// TwinCAT 3 PLC project LightSwitch
// ProgramVersion: 3.1.4023.0
// libraries:
//   Tc2_Standard, * (Beckhoff Automation GmbH)
//   Tc2_System, * (Beckhoff Automation GmbH)
//   Tc3_Module, * (Beckhoff Automation GmbH)
// project tree:
//   / PlcTask.TcTTO
//   POUs/Customer/ FB_LightController.TcPOU
//   POUs/Lib/ FB_LightBase.TcPOU, FB_LightDimmable.TcPOU, FB_LightGroup.TcPOU, I_LightBase.TcIO, I_LightDimmable.TcIO
//   POUs/ MAIN.TcPOU
// real-time tasks:
//   TASK PlcTask1: cycle T#10ms, priority 21, ADS port 351

CONFIGURATION LightSwitch
    RESOURCE PLC ON TwinCAT3
        TASK PlcTask(INTERVAL := T#10ms, PRIORITY := 21);
        PROGRAM MAIN WITH PlcTask : MAIN;
    END_RESOURCE
END_CONFIGURATION

// ---- POUs/Lib/I_LightBase.TcIO
INTERFACE I_LightBase EXTENDS __SYSTEM.IQueryInterface

PROPERTY ID : USINT
GET
END_GET
SET
END_SET
END_PROPERTY

PROPERTY PUBLIC State : BOOL
GET
END_GET
SET
END_SET
END_PROPERTY

METHOD Toggle
END_METHOD

METHOD TurnOFF
END_METHOD

METHOD TurnON
END_METHOD

END_INTERFACE

// ---- POUs/Lib/I_LightDimmable.TcIO
INTERFACE I_LightDimmable EXTENDS I_LightBase

PROPERTY Brightness : USINT
GET
END_GET
SET
END_SET
END_PROPERTY

END_INTERFACE

// ---- POUs/MAIN.TcPOU
PROGRAM MAIN
VAR
	fbLightController	: FB_LightController;
END_VAR
VAR CONSTANT
	MAXIMUM_NUMBER_OF_LIGHTS	: USINT := 8;
END_VAR

fbLightController();

END_PROGRAM

// ---- POUs/Customer/FB_LightController.TcPOU
FUNCTION_BLOCK FB_LightController
VAR
	_iLight									: I_LightBase;
	_iLightB								: I_LightDimmable;
	                    	    			
	fbLightGroup							: FB_LightGroup;
	                    	    			
	fbLightBase_1							: FB_LightBase;
	fbLightBase_2							: FB_LightBase;
	fbLightBase_3							: FB_LightBase;
	fbLightBase_4							: FB_LightBase;
	fbLightDimmable_5						: FB_LightDimmable;
	fbLightDimmable_6						: FB_LightDimmable;
	fbLightDimmable_7						: FB_LightDimmable;
	fbLightDimmable_8						: FB_LightDimmable;
	                    	    			
	nBrightness								: USINT := 100;
	                    	    			
	bToggle									: BOOL;
	bSwitch									: BOOL;
	bSetBrightness							: BOOL;
	                    	    			
	tToggle									: R_TRIG;
	tSwitchON								: R_TRIG;
	tSwitchOFF								: F_TRIG;
	tSetBrightness							: R_TRIG;
	                    	    			
	bGroupSwitch							: BOOL;
	bSetGroupBrightness						: BOOL;
	                    	    			
	tGroupSwitchON							: R_TRIG;
	tGroupSwitchOFF							: F_TRIG;
	tSetGroupBrightness						: R_TRIG;
	                    	    			
	eSwitchOptions							: (WAIT, TOGGLE, SWITCHON, SWITCHOFF, SETBRIGHTNESS, GROUPSWITCHON, GROUPSWITCHOFF, SETGROUPBRIGHTNESS);
	
	eSwitchControlledLightObjectByLightID	: (LIGHT_ONE, LIGHT_TWO, LIGHT_THREE, LIGHT_FOUR, LIGHT_FIVE, LIGHT_SIX, LIGHT_SEVEN, LIGHT_EIGHT);

END_VAR

fbLightGroup();

CASE eSwitchOptions OF
	WAIT:
		//do nothing
	TOGGLE:
		_iLight.Toggle();
		eSwitchOptions := WAIT;
	SWITCHON:
		_iLight.TurnON();
		eSwitchOptions := WAIT;
	SWITCHOFF:
		_iLight.TurnOFF();
		eSwitchOptions := WAIT;
	SETBRIGHTNESS:
		IF __QUERYINTERFACE(_iLight, _iLightB) THEN
			_iLightB.Brightness := nBrightness;	
		END_IF
		eSwitchOptions := WAIT;
	GROUPSWITCHON:
		fbLightGroup.TurnON();
		eSwitchOptions := WAIT;
	GROUPSWITCHOFF:
		fbLightGroup.TurnOFF();
		eSwitchOptions := WAIT;
	SETGROUPBRIGHTNESS:
		fbLightGroup.SetBrightness(nBrightness);
		eSwitchOptions := WAIT;
END_CASE

CASE eSwitchControlledLightObjectByLightID OF
	LIGHT_ONE:
		ipLight := fbLightBase_1;
	LIGHT_TWO:
		ipLight := fbLightBase_2;
	LIGHT_THREE:
		ipLight := fbLightBase_3;
	LIGHT_FOUR:
		ipLight := fbLightBase_4;
	LIGHT_FIVE:
		ipLight := fbLightDimmable_5;
	LIGHT_SIX:
		ipLight := fbLightDimmable_6;
	LIGHT_SEVEN:
		ipLight := fbLightDimmable_7;
	LIGHT_EIGHT:
		ipLight := fbLightDimmable_8;
END_CASE

tToggle(CLK := bToggle);
tSwitchON(CLK := bSwitch);
tSwitchOFF(CLK := bSwitch);
tSetBrightness(CLK := bSetBrightness);

tGroupSwitchOFF(CLK := bGroupSwitch);
tGroupSwitchON(CLK := bGroupSwitch);
tSetGroupBrightness(CLK := bSetGroupBrightness);

IF tToggle.Q THEN
	eSwitchOptions := TOGGLE;
	bToggle := FALSE;									
END_IF

IF tSwitchON.Q THEN
	eSwitchOptions := SWITCHON;
END_IF

IF tSwitchOFF.Q THEN
	eSwitchOptions := SWITCHOFF;
END_IF

IF tSetBrightness.Q THEN
	eSwitchOptions := SETBRIGHTNESS;
	bSetBrightness := FALSE;
END_IF

IF tGroupSwitchON.Q THEN
	eSwitchOptions := GROUPSWITCHON;
END_IF

IF tGroupSwitchOFF.Q THEN
	eSwitchOptions := GROUPSWITCHOFF;
END_IF

IF tSetGroupBrightness.Q THEN
	eSwitchOptions := SETGROUPBRIGHTNESS;
	bSetGroupBrightness := FALSE;
END_IF

METHOD FB_init : BOOL
VAR_INPUT
	bInitRetains	: BOOL; // if TRUE, the retain variables are initialized (warm start / cold start)
	bInCopyCode		: BOOL;  // if TRUE, the instance afterwards gets moved into the copy code (online change)
END_VAR
_iLight := fbLightBase_1;

fbLightGroup.ImportLight(fbLightBase_1);
fbLightGroup.ImportLight(fbLightBase_2);
fbLightGroup.ImportLight(fbLightBase_3);
fbLightGroup.ImportLight(fbLightBase_4);
fbLightGroup.ImportLight(fbLightDimmable_5);
fbLightGroup.ImportLight(fbLightDimmable_6);
fbLightGroup.ImportLight(fbLightDimmable_7);
fbLightGroup.ImportLight(fbLightDimmable_8);
END_METHOD

PROPERTY ipLight : I_LightBase
GET
ipLight := _iLight;
END_GET
SET
_iLight := ipLight;
END_SET
END_PROPERTY

END_FUNCTION_BLOCK

// ---- POUs/Lib/FB_LightGroup.TcPOU
FUNCTION_BLOCK FB_LightGroup
VAR
	CurrentSizeOfLightGroup		: USINT := 0;
	aLights						: ARRAY[0..MAIN.MAXIMUM_NUMBER_OF_LIGHTS-1] OF I_LightBase;
	nCounter					: USINT;
	
	bIsOn						: bool := false;
END_VAR

// import all lights from main

FOR nCounter := 0 TO CurrentSizeOfLightGroup - 1 DO
	IF aLights[nCounter].State THEN
		bIsOn := TRUE;
		EXIT;
	ELSE
		IF nCounter = CurrentSizeOfLightGroup - 1 THEN
			bIsOn := FALSE;
		END_IF
	END_IF
END_FOR

METHOD ImportLight : BOOL
VAR_INPUT
	iLight		: I_LightBase;
END_VAR
aLights[CurrentSizeOfLightGroup]	:= iLight;
CurrentSizeOfLightGroup := CurrentSizeOfLightGroup + 1;
iLight.ID := CurrentSizeOfLightGroup;
END_METHOD

METHOD SetBrightness
VAR_INPUT
	nBrightness	: USINT;
END_VAR
VAR
	nCounter: USINT;
	iBrightness	: I_LightDimmable;
END_VAR
IF aLights[nCounter] <> 0 THEN
	FOR nCounter := 0 TO CurrentSizeOfLightGroup-1 DO
		IF __QUERYINTERFACE(aLights[nCounter], iBrightness) THEN
			iBrightness.Brightness := nBrightness;
		END_IF
	END_FOR
END_IF
END_METHOD

METHOD TurnOFF
VAR
	nCounter	: USINT;
END_VAR
FOR nCounter := 0 TO CurrentSizeOfLightGroup-1	DO
	aLights[nCounter].State := FALSE;
END_FOR
END_METHOD

METHOD TurnON
VAR
	nCounter	: USINT;
END_VAR
FOR nCounter := 0 TO CurrentSizeOfLightGroup-1	DO
	aLights[nCounter].State := TRUE;
END_FOR
END_METHOD

END_FUNCTION_BLOCK

// ---- POUs/Lib/FB_LightBase.TcPOU
FUNCTION_BLOCK FB_LightBase IMPLEMENTS I_LightBase

VAR
	sName				: STRING;
	sAddress			: STRING;
	bState				: BOOL;
	nLightID			: USINT;
END_VAR

PROPERTY ID : USINT
GET
ID := nLightID;
END_GET
SET
nLightID := ID;
END_SET
END_PROPERTY

PROPERTY PUBLIC State : BOOL
GET
State := bState;
END_GET
SET
bState := State;
END_SET
END_PROPERTY

METHOD Toggle
IF NOT bState THEN
	THIS^.TurnON();
ELSE
	THIS^.TurnOFF();
END_IF
END_METHOD

METHOD TurnOFF
THIS^.bState := FALSE;
END_METHOD

METHOD TurnON
THIS^.bState := TRUE;
END_METHOD

END_FUNCTION_BLOCK

// ---- POUs/Lib/FB_LightDimmable.TcPOU
FUNCTION_BLOCK FB_LightDimmable EXTENDS FB_LightBase IMPLEMENTS I_LightDimmable
VAR
	nBrightness	: USINT := 100;
END_VAR

PROPERTY PUBLIC Brightness : USINT;
GET
Brightness := nBrightness;
END_GET
SET
nBrightness := Brightness;
END_SET
END_PROPERTY

END_FUNCTION_BLOCK
